Universal Robots PolyScope program: tercero.urp

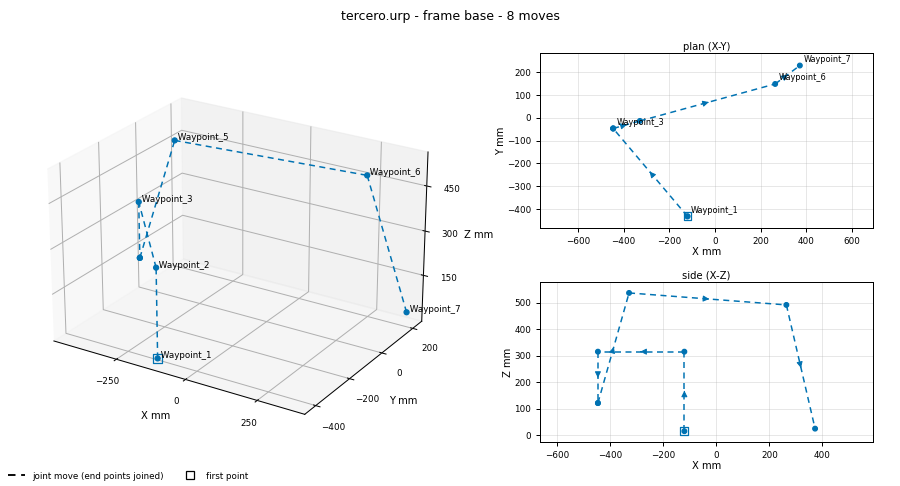
[picture p0: tool path of tercero.urp in frame base, 8 of 8 moves have a stored position in this frame; points joined in program order, loops and branches not executed]
Program tercero (installation=default directory=/ursim/programs createdIn=3.15.8.106339 lastSavedIn=3.15.8.106339 robotSerialNumber=2018359999)
Calibrated DH parameters: a=[0, -0.425, -0.39225, 0, 0, 0]; d=[0.089159, 0, 0, 0.10915, 0.09465, 0.0823]; alpha=[1.570796, 0, 0, 1.570796, -1.570796, 0]; deltaTheta=[0, 0, 0, 0, 0, 0]
Robot Program (runOnlyOnce=false)
  Popup Message (haltProgram=false message=Primera posición y se activa el efector final inputType=Text)
  Set DigitalOutput pin=digital_out[0]; digitalValue=1
  Wait Sleep waitTime=1
  MoveJ speed 60 deg/s, acceleration 80 deg/s^2 (useActiveTCP=true)
    Waypoint Waypoint_1: TCP in base x=-120.113 y=-431.763 z=16.154 mm, rx=-0.0012 ry=3.1163 rz=0.0389 rad; joints [-91.713, -117.731, -130.591, -23.151, 91.393, -1.776] deg
    Waypoint Waypoint_2: TCP in base x=-120.113 y=-431.763 z=315.751 mm, rx=-0.0012 ry=3.1163 rz=0.0389 rad; joints [-91.713, -85.529, -111.128, -74.816, 91.393, -1.776] deg
    Waypoint Waypoint_3: TCP in base x=-445.726 y=-46.638 z=315.751 mm, rx=1.7471 ry=2.569 rz=0.0101 rad; joints [-160.194, -85.529, -111.128, -74.816, 91.393, -1.776] deg
    Waypoint Waypoint_4: TCP in base x=-445.726 y=-46.638 z=122.152 mm, rx=1.7471 ry=2.569 rz=0.0101 rad; joints [-160.194, -101.92, -127.555, -41.998, 91.393, -1.776] deg
    Set DigitalOutput pin=digital_out[0]; digitalValue=0
    Wait Sleep waitTime=1
    Popup Message (haltProgram=false message=Se libera el objeto y se recoge el otro inputType=Text)
  Set DigitalOutput pin=digital_out[0]; digitalValue=1
  MoveJ speed 60 deg/s, acceleration 80 deg/s^2 (useActiveTCP=true)
    Waypoint Waypoint_4: TCP in base x=-445.726 y=-46.638 z=122.152 mm, rx=1.7471 ry=2.569 rz=0.0101 rad; joints [-160.194, -101.92, -127.555, -41.998, 91.393, -1.776] deg
    Waypoint Waypoint_5: TCP in base x=-328.42 y=-13.555 z=536.975 mm, rx=-1.6281 ry=-2.4074 rz=0.4853 rad; joints [-158.622, -64.145, -100.13, -83.783, 91.432, -0.204] deg
    Waypoint Waypoint_6: TCP in base x=264.155 y=148.386 z=491.833 mm, rx=2.9253 ry=-1.059 rz=-0.0585 rad; joints [-309.976, -64.145, -100.13, -108.077, 91.432, -0.204] deg
    Waypoint Waypoint_7: TCP in base x=372.321 y=229.195 z=25.789 mm, rx=2.7568 ry=-0.9801 rz=0.4683 rad; joints [-309.976, -115.28, -133.259, -24.915, 69.43, -0.204] deg
    Set DigitalOutput pin=digital_out[0]; digitalValue=0
    Wait Sleep waitTime=1
    Popup Message (haltProgram=false message=Se libera el segundo objeto inputType=Text)
  Wait DigitalInput pin=digital_in[0]; digitalValue=1
